{attribute 'qualified_only'}
VAR_GLOBAL
	test1: BOOL;
END_VAR

(* stored: Version 1.1.0.1, ProductVersion 3.1.4024.11
   GVL GVLtest1: Id {71dbad84-4e7d-4ced-9ca7-6429e7799d7b} *)
